FUNCTION_BLOCK PUBLIC FB_RunControl
VAR
	statRuncontrolActive	:	BOOL;
END_VAR

METHOD PUBLIC ActivateRunControl
VAR_INPUT
	Activate	:	BOOL;
END_VAR
IF Activate	THEN
	statRuncontrolActive := TRUE;
END_IF
END_METHOD

METHOD PUBLIC DeactivateRunControl
VAR_INPUT
	Deactivate	:	BOOL;
END_VAR
IF Deactivate THEN
	statRuncontrolActive := FALSE;
END_IF
END_METHOD

PROPERTY PUBLIC IsActive : BOOL
GET
IsActive := statRuncontrolActive;
END_GET
END_PROPERTY

END_FUNCTION_BLOCK

(* stored: Version 1.1.0.1
   POU FB_RunControl: Id {ca2eaa5d-b744-4f82-9238-240684bd257a}, SpecialFunc None
   Method ActivateRunControl: Id {34162a8a-9518-40b6-9439-52e0599e4c5b}
   Method DeactivateRunControl: Id {00b61f17-8e7a-4b0f-9b26-56c7cea82755}
   Property IsActive: Id {e89aaee9-99a8-4638-b76b-de6f9adebe2c}
   Get Get: Id {42b13b13-458a-4c0b-a357-1400f6782730} *)
